Fanuc KAREL source: kb00060.KL

-- PROVISIONAL review KL for V940-1; original PC SHA256 6e18c5785d7eba6488b59dee261562e02fecf97f8a57f61c0cdc2be7cf9b6cc3
-- Incomplete behavior may be omitted. Consult companion uncertainty JSON. Do not deploy.
PROGRAM KB00060
%NOLOCKGROUP
BEGIN
  -- V9_ZERO_TABLE_METADATA_HINT layout=0002_ascii; no indexed target words; source/name/runtime held
  -- UNRESOLVED_PC offsets 5-14; opcodes 3F,75
  -- UNRESOLVED_PC offsets 19-26; opcodes 9D,23
  -- UNRESOLVED_PC offsets 31-38; opcodes 9D,23
  -- UNRESOLVED_PC offsets 43-50; opcodes 9D,23
  -- UNRESOLVED_PC offsets 55-62; opcodes 9D,23
  -- UNRESOLVED_PC offsets 67-103; opcodes 27,22,2A,22,22,22,22,31
  -- UNRESOLVED_PC offsets 108-112; opcodes 7F
END KB00060
